// TIA Portal V19 export
TYPE "UDT_AINWARNS"
   STRUCT
      ctrl : Struct   // External data (Primary warning data - alarm & plc ackn)
         alarm_h : Bool := false;
         alarm_l : Bool := false;
         bit10 : Bool := false;
         bit11 : Bool := false;
         bit12 : Bool := false;
         bit13 : Bool := false;
         bit14 : Bool := false;
         bit15 : Bool := false;
         plcackn_h : Bool := false;
         plcackn_l : Bool := false;
         plcackn_over : Bool := false;
         plcackn_under : Bool := false;
         bit4 : Bool := false;
         bit5 : Bool := false;
         bit6 : Bool := false;
         bit7 : Bool := false;
      END_STRUCT;
      status : Struct   // External data (Secondary warning data - siren & hmi ackn)
         siren_h : Bool := false;
         siren_l : Bool := false;
         bit10 : Bool := false;
         bit11 : Bool := false;
         bit12 : Bool := false;
         bit13 : Bool := false;
         bit14 : Bool := false;
         bit15 : Bool := false;
         hmiackn_h : Bool := false;
         hmiackn_l : Bool := false;
         hmiackn_over : Bool := false;
         hmiackn_under : Bool := false;
         bit4 : Bool := false;
         bit5 : Bool := false;
         bit6 : Bool := false;
         bit7 : Bool := false;
      END_STRUCT;
   END_STRUCT;
END_TYPE
